// TIA Portal project "PLC2_Cell" (V19)

(* hardware
DEVICE "S7-1200 station_1"  S7-1200 Station
   slot 0: "Rack_0"  S7-1200 Rack  Rack  V1.0
   slot 1: "PLC_Machining"  CPU 1214C AC/DC/Rly  6ES7 214-1BG40-0XB0  V4.5
   slot 2: "DI 16x24VDC/DQ 16xRelay_1"  SM 1223 DI16/DQ16 x relay  6ES7 223-1PL32-0XB0  V2.0
   slot 3: "AQ 1x12BIT_1"  AQ1 signal board  6ES7 232-4HA30-0XB0  V1.0
   slot 3: "AI 4x13BIT/AQ 2x14BIT_1"  6ES7 234-4HE32-0XB0  V2.1
DEVICE "HMI_1"  KTP700 Basic PN
   slot 0: "HMI_1"  KTP700 Basic PN  6AV2 123-2GB03-0AX0  17.0.0.0
   slot 1: "HMI_RT_1"  KTP700 Basic PN  6AV2 123-2GB03-0AX0  17.0.0.0
   slot 5: "HMI_1.IE_CP_1"  PROFINET Interface  17.0.0.0
      slot 1: "PROFINET Interface_1"  PROFINET Interface
         slot 1: "Port_1"  Port
DEVICE "S7-1200 station_2"  S7-1200 Station
   slot 0: "Rack_0"  S7-1200 Rack  Rack  V1.0
   slot 1: "PLC_Pneumatic"  CPU 1214C AC/DC/Rly  6ES7 214-1BG40-0XB0  V4.5
   slot 2: "DI 16x24VDC/DQ 16xRelay_1"  SM 1223 DI16/DQ16 x relay  6ES7 223-1PL32-0XB0  V2.0
   slot 3: "AQ 1x12BIT_1"  AQ1 signal board  6ES7 232-4HA30-0XB0  V1.0
   slot 3: "AI 4x13BIT/AQ 2x14BIT_1"  6ES7 234-4HE32-0XB0  V2.1
DEVICE "HMI_2"  KTP700 Basic PN
   slot 0: "HMI_2"  KTP700 Basic PN  6AV2 123-2GB03-0AX0  17.0.0.0
   slot 1: "HMI_RT_2"  KTP700 Basic PN  6AV2 123-2GB03-0AX0  17.0.0.0
   slot 5: "HMI_2.IE_CP_1"  PROFINET Interface  17.0.0.0
      slot 1: "PROFINET Interface_1"  PROFINET Interface
         slot 1: "Port_1"  Port
*)

// ===== PLC "PLC_Machining"  CPU 1214C AC/DC/Rly =====

VAR_GLOBAL   // PLC tag table "Default tag table"
   "Pusher_latch" AT %M10.0 : Bool;
   "Conveyor2_latch" AT %M10.1 : Bool;
   "Conveyor4_latch" AT %M10.2 : Bool;
   "Conveyor3_latch" AT %M10.3 : Bool;
   "Conveyor5_latch" AT %M10.4 : Bool;
   "Conveyor6_IN_latch" AT %M10.5 : Bool;
   "Conveyor6_OUT_latch" AT %M10.6 : Bool;
   "Conveyor6_Position" AT %M10.7 : Bool;
   "lampBlinkTag" AT %M11.0 : Bool;
   "cakeFlavor" AT %MW12 : UInt;
   "drillingTime" AT %MD14 : Time;
   "mixingTime" AT %MD18 : Time;
   "System_Byte" AT %MB22 : Byte;
   "FirstScan" AT %M22.0 : Bool;
   "DiagStatusUpdate" AT %M22.1 : Bool;
   "AlwaysTRUE" AT %M22.2 : Bool;
   "AlwaysFALSE" AT %M22.3 : Bool;
   "drillActive" AT %M23.0 : Bool;
   "mixActive" AT %M23.1 : Bool;
   "CognexCode" AT %MW24 : Int;
END_VAR

VAR_GLOBAL   // PLC tag table "Cell_Tags"
   "Opto_Conveyor6B" AT %I8.0 : Bool;
   "Press_BTN_DOWN" AT %I8.2 : Bool;
   "Conveyor2" AT %Q0.0 : Bool;
   "Pusher1" AT %Q0.1 : Bool;
   "Conveyor4" AT %Q0.4 : Bool;
   "Conveyor5" AT %Q0.7 : Bool;
   "Conveyor3" AT %Q0.2 : Bool;
   "Drill" AT %Q0.3 : Bool;
   "Mix" AT %Q0.5 : Bool;
   "Pusher2" AT %Q0.6 : Bool;
   "Green_Tower" AT %Q1.0 : Bool;
   "Red_Tower" AT %Q1.1 : Bool;
   "Conveyor6_OUT" AT %Q8.3 : Bool;
   "Press_UP" AT %Q8.4 : Bool;
   "Press_DOWN" AT %Q8.5 : Bool;
   "Conveyor6_IN" AT %Q8.2 : Bool;
   "Press_BTN_UP" AT %I8.3 : Bool;
   "Opto_Conveyor2A" AT %I0.0 : Bool;
   "Opto_Conveyor2B" AT %I0.1 : Bool;
   "Green_Light" AT %Q9.5 : Bool;
   "Red_Light" AT %Q9.6 : Bool;
   "Blue_Light" AT %Q9.7 : Bool;
   "Green_BTN" AT %I9.4 : Bool;
   "Yellow_BTN" AT %I9.5 : Bool;
   "Red_BTN" AT %I9.6 : Bool;
   "Emergency_BTN" AT %I9.7 : Bool;
   "Pusher1_BTN" AT %I0.2 : Bool;
   "Opto_Drill" AT %I0.3 : Bool;
   "Opto_Mix" AT %I0.4 : Bool;
   "Opto_Conveyor5" AT %I0.6 : Bool;
   "Pusher2_BTN" AT %I0.5 : Bool;
   "Opto_Conveyor6A" AT %I8.1 : Bool;
   "Conveyor2_tactileSW" AT %I0.7 : Bool;
   "cellPotentiometer" AT %IW64 : Int;
   "AO_Channel0" AT %QW112 : Int;
   "AO_Channel1" AT %QW114 : Int;
   "AO_Cell" AT %QW80 : Int;
   "Cognex_out0" AT %I9.0 : Bool;
   "Cognex_out1" AT %I9.1 : Bool;
   "Cognex_out2" AT %I9.2 : Bool;
   "Cognex_in0" AT %Q8.7 : Bool;
END_VAR

VAR_GLOBAL   // PLC tag table "HMI_Tags"
   "HMI_BTN1" AT %M50.0 : Bool;
   "HMI_BTN_Conveyor2" AT %M50.1 : Bool;
   "HMI_BTN_Pusher1" AT %M50.2 : Bool;
   "HMI_BTN_Conveyor3" AT %M50.3 : Bool;
   "HMI_BTN_Conveyor4" AT %M50.4 : Bool;
   "HMI_BTN_Conveyor5" AT %M50.5 : Bool;
   "HMI_BTN_Drill" AT %M50.6 : Bool;
   "HMI_BTN_Mix" AT %M50.7 : Bool;
   "HMI_BTN_Pusher2" AT %M51.0 : Bool;
   "HMI_BTN10" AT %M51.1 : Bool;
   "HMI_BTN11" AT %M51.2 : Bool;
   "HMI_BTN12" AT %M51.3 : Bool;
   "HMI_BTN13" AT %M51.4 : Bool;
   "HMI_BTN14" AT %M51.5 : Bool;
   "HMI_BTN15" AT %M51.6 : Bool;
   "HMI_BTN16" AT %M51.7 : Bool;
   "HMI_BTN17" AT %M52.0 : Bool;
   "HMI_BTN18" AT %M52.1 : Bool;
   "HMI_BTN19" AT %M52.2 : Bool;
   "HMI_BTN20" AT %M52.3 : Bool;
   "HMI_BTN21" AT %M52.4 : Bool;
   "HMI_BTN22" AT %M52.5 : Bool;
   "HMI_BTN23" AT %M52.6 : Bool;
   "HMI_BTN24" AT %M52.7 : Bool;
   "ManualMode_SW" AT %M53.0 : Bool;
END_VAR

VAR_GLOBAL   // PLC tag table "Clock_Memory_Tags"
   "Clock_Byte" AT %MB0 : Byte;
   "Clock_10Hz" AT %M0.0 : Bool;
   "Clock_5Hz" AT %M0.1 : Bool;
   "Clock_2.5Hz" AT %M0.2 : Bool;
   "Clock_2Hz" AT %M0.3 : Bool;
   "Clock_1.25Hz" AT %M0.4 : Bool;
   "Clock_1Hz" AT %M0.5 : Bool;
   "Clock_0.625Hz" AT %M0.6 : Bool;
   "Clock_0.5Hz" AT %M0.7 : Bool;
END_VAR

DATA_BLOCK "potentiometerValue"   // DB14
{ S7_Optimized_Access := 'TRUE' }
VERSION : 0.1
// stored: InstanceOfName FB_AnalogInput
"FB_AnalogInput"
BEGIN
END_DATA_BLOCK

DATA_BLOCK "processTimes_DB"   // DB15
{ S7_Optimized_Access := 'TRUE' }
VERSION : 0.1
   VAR
      chocolateDrillingInput_ms : UInt := 3000;
      chocolateMixingInput_ms : UInt := 3000;
      vanillaDrillingInput_ms : UInt := 5000;
      vanillaMixingInput_ms : UInt := 5000;
      strawberryDrillingInput_ms : UInt := 7000;
      strawberryMixingInput_ms : UInt := 7000;
      chocolateDrilling_s : Time;
      chocolateMixing_s : Time;
      vanillaDrilling_s : Time;
      vanillaMixing_s : Time;
      strawberryDrilling_s : Time;
      strawberryMixing_s : Time;
   END_VAR
BEGIN
END_DATA_BLOCK

DATA_BLOCK "Machining_Communication_DB"   // DB100
{ S7_Optimized_Access := 'FALSE' }
VERSION : 0.1
   VAR
      Cognex_Code : Int;   // Machining to Pneu
      Cobot_Code : Int;   // Pneu to Machining
      Cake_ID : Int;   // Pneu to Machining
      EmergencyStop : Bool;
      Cognex_Shutter : Bool;   // Pneu to Machining
      Conveyor5_Done : Bool;   // Machining to Pneu
      Conveyor6_Done : Bool;   // Machining to Pneu
      Conveyor1_Sensor : Bool;   // Pneu to Machining
      Conveyor2_SensorA : Bool;   // Machining to Pneu
   END_VAR
BEGIN
END_DATA_BLOCK

// folder: System blocks/Program resources

DATA_BLOCK "Mix_PostTP"   // DB1
{ S7_Optimized_Access := 'TRUE' }
AUTHOR : Simatic
FAMILY : IEC
NAME : IEC_TMR
VERSION : 1.0
// stored: InstanceOfName IEC_TIMER
"IEC_TIMER"
BEGIN
END_DATA_BLOCK

DATA_BLOCK "Pusher1_Delay"   // DB2
{ S7_Optimized_Access := 'TRUE' }
AUTHOR : Simatic
FAMILY : IEC
NAME : IEC_TMR
VERSION : 1.0
// stored: InstanceOfName IEC_TIMER
"IEC_TIMER"
BEGIN
END_DATA_BLOCK

DATA_BLOCK "Drill_OperationTP"   // DB3
{ S7_Optimized_Access := 'TRUE' }
AUTHOR : Simatic
FAMILY : IEC
NAME : IEC_TMR
VERSION : 1.0
// stored: InstanceOfName IEC_TIMER
"IEC_TIMER"
BEGIN
END_DATA_BLOCK

DATA_BLOCK "Mix_OperationTP"   // DB4
{ S7_Optimized_Access := 'TRUE' }
AUTHOR : Simatic
FAMILY : IEC
NAME : IEC_TMR
VERSION : 1.0
// stored: InstanceOfName IEC_TIMER
"IEC_TIMER"
BEGIN
END_DATA_BLOCK

DATA_BLOCK "Drill_PostTP"   // DB5
{ S7_Optimized_Access := 'TRUE' }
AUTHOR : Simatic
FAMILY : IEC
NAME : IEC_TMR
VERSION : 1.0
// stored: InstanceOfName IEC_TIMER
"IEC_TIMER"
BEGIN
END_DATA_BLOCK

DATA_BLOCK "Conveyor2_TP"   // DB6
{ S7_Optimized_Access := 'TRUE' }
AUTHOR : Simatic
FAMILY : IEC
NAME : IEC_TMR
VERSION : 1.0
// stored: InstanceOfName IEC_TIMER
"IEC_TIMER"
BEGIN
END_DATA_BLOCK

DATA_BLOCK "Conveyor2_ManualDelay"   // DB7
{ S7_Optimized_Access := 'TRUE' }
AUTHOR : Simatic
FAMILY : IEC
NAME : IEC_TMR
VERSION : 1.0
// stored: InstanceOfName IEC_TIMER
"IEC_TIMER"
BEGIN
END_DATA_BLOCK

DATA_BLOCK "Pusher2_Delay"   // DB8
{ S7_Optimized_Access := 'TRUE' }
AUTHOR : Simatic
FAMILY : IEC
NAME : IEC_TMR
VERSION : 1.0
// stored: InstanceOfName IEC_TIMER
"IEC_TIMER"
BEGIN
END_DATA_BLOCK

DATA_BLOCK "Press_Delay"   // DB9
{ S7_Optimized_Access := 'TRUE' }
AUTHOR : Simatic
FAMILY : IEC
NAME : IEC_TMR
VERSION : 1.0
// stored: InstanceOfName IEC_TIMER
"IEC_TIMER"
BEGIN
END_DATA_BLOCK

DATA_BLOCK "IEC_Timer_0_DB"   // DB10
{ S7_Optimized_Access := 'TRUE' }
AUTHOR : Simatic
FAMILY : IEC
NAME : IEC_TMR
VERSION : 1.0
// stored: InstanceOfName IEC_TIMER
"IEC_TIMER"
BEGIN
END_DATA_BLOCK

DATA_BLOCK "Press_DOWN_Timer"   // DB11
{ S7_Optimized_Access := 'TRUE' }
AUTHOR : Simatic
FAMILY : IEC
NAME : IEC_TMR
VERSION : 1.0
// stored: InstanceOfName IEC_TIMER
"IEC_TIMER"
BEGIN
END_DATA_BLOCK

DATA_BLOCK "Emergency_Blink_TP"   // DB12
{ S7_Optimized_Access := 'TRUE' }
AUTHOR : Simatic
FAMILY : IEC
NAME : IEC_TMR
VERSION : 1.0
// stored: InstanceOfName IEC_TIMER
"IEC_TIMER"
BEGIN
END_DATA_BLOCK

DATA_BLOCK "Emergency_Blink_TON"   // DB13
{ S7_Optimized_Access := 'TRUE' }
AUTHOR : Simatic
FAMILY : IEC
NAME : IEC_TMR
VERSION : 1.0
// stored: InstanceOfName IEC_TIMER
"IEC_TIMER"
BEGIN
END_DATA_BLOCK

// folder: (top level)

FUNCTION_BLOCK "FB_AnalogInput"   // FB1, LAD
{ S7_Optimized_Access := 'TRUE' }
VERSION : 0.1
   VAR_INPUT
      minRaw : Int;
      maxRaw : Int := 27648;
      rawValue : Int;
      minScale : Real;
      maxScale : Real := 1.0;
   END_VAR
   VAR_OUTPUT
      outputValue : Real;
   END_VAR
   VAR_TEMP
      normValue : Real;
   END_VAR
BEGIN

REGION Network 1
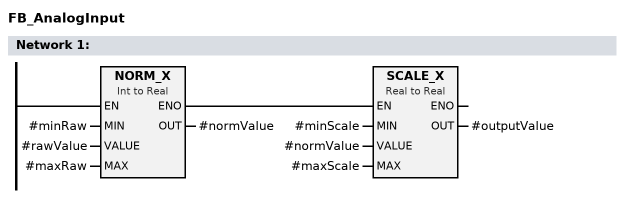
   RUNG wire#powerrail
      { S7_Templates := "[SrcType := Int, DestType := Real]" } Normalize(min := #minRaw, value := #rawValue, max := #maxRaw, out => #normValue)
      { S7_Templates := "[SrcType := Real, DestType := Real]" } Scale(min := #minScale, value := #normValue, max := #maxScale, out => #outputValue)
   END_RUNG
   // the same network as SCL:
   #normValue := NORM_X(MIN := #minRaw, VALUE := #rawValue, MAX := #maxRaw);
   #outputValue := SCALE_X(MIN := #minScale, VALUE := #normValue, MAX := #maxScale);
END_REGION
END_FUNCTION_BLOCK

ORGANIZATION_BLOCK "Main"   // OB1, LAD, ProgramCycle
TITLE = "Main Program Sweep (Cycle)"
{ S7_Optimized_Access := 'TRUE' }
VERSION : 0.1
   VAR_INPUT
      Initial_Call : Bool;   // Initial call of this OB
      Remanence : Bool;   // =True, if remanent data are available
   END_VAR
   VAR_TEMP   // added for the SCL form of the ladder/FBD networks
      _w1 : Bool;
   END_VAR
BEGIN

REGION Network 1: Conveyor #2
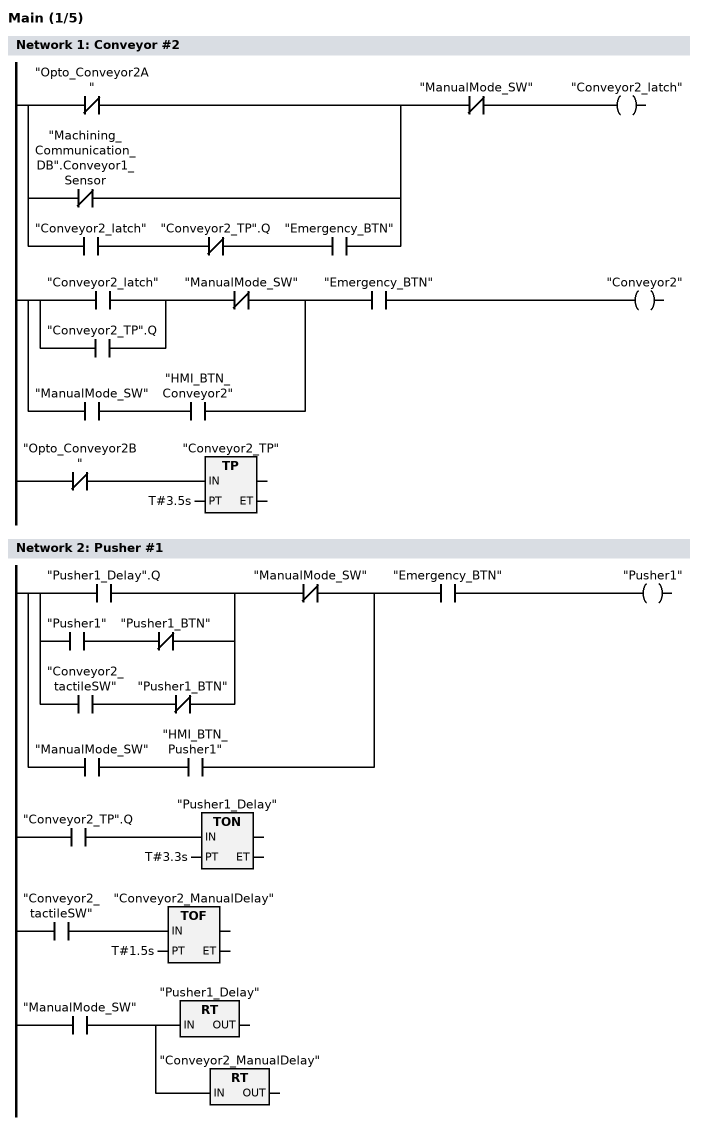
   "Conveyor2_latch" := (NOT "Opto_Conveyor2A" OR NOT "Machining_Communication_DB".Conveyor1_Sensor OR ("Conveyor2_latch" AND NOT "Conveyor2_TP".Q AND "Emergency_BTN")) AND NOT "ManualMode_SW";
   "Conveyor2" := ((("Conveyor2_latch" OR "Conveyor2_TP".Q) AND NOT "ManualMode_SW") OR ("ManualMode_SW" AND "HMI_BTN_Conveyor2")) AND "Emergency_BTN";
   "Conveyor2_TP".TP(IN := NOT "Opto_Conveyor2B", PT := T#3.5s);
END_REGION

REGION Network 2: Pusher #1
   "Pusher1" := ((("Pusher1_Delay".Q OR ("Pusher1" AND NOT "Pusher1_BTN") OR ("Conveyor2_tactileSW" AND NOT "Pusher1_BTN")) AND NOT "ManualMode_SW") OR ("ManualMode_SW" AND "HMI_BTN_Pusher1")) AND "Emergency_BTN";
   "Pusher1_Delay".TON(IN := "Conveyor2_TP".Q, PT := T#3.3s);
   "Conveyor2_ManualDelay".TOF(IN := "Conveyor2_tactileSW", PT := T#1.5s);
   IF "ManualMode_SW" THEN
       RESET_TIMER("Pusher1_Delay");
       RESET_TIMER("Conveyor2_ManualDelay");
   END_IF;
END_REGION

REGION Network 3: Conveyor 3: Drill
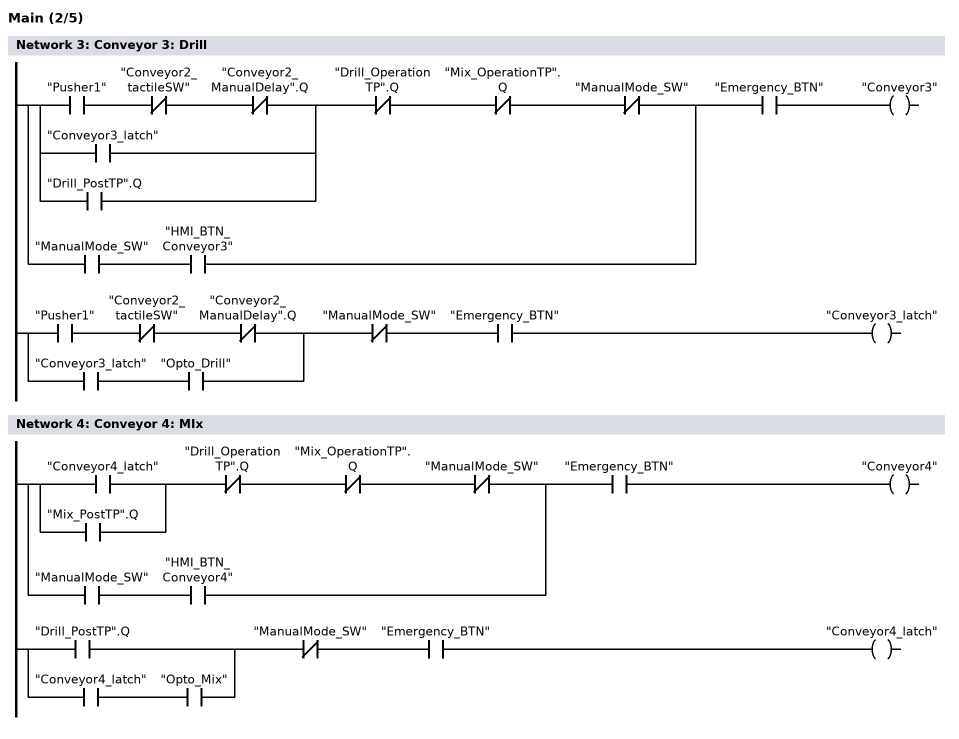
   RUNG wire#powerrail
      Contact( "Pusher1" )
      I_Contact( "Conveyor2_tactileSW" )
      I_Contact( "Conveyor2_ManualDelay".Q )
      wire#w1
      I_Contact( "Drill_OperationTP".Q )
      I_Contact( "Mix_OperationTP".Q )
      I_Contact( "ManualMode_SW" )
      wire#w2
      Contact( "Emergency_BTN" )
      Coil( "Conveyor3" )
   END_RUNG
   RUNG wire#powerrail
      Contact( "Conveyor3_latch" )
   END_RUNG wire#w1
   RUNG wire#powerrail
      Contact( "Drill_PostTP".Q )
   END_RUNG wire#w1
   RUNG wire#powerrail
      Contact( "ManualMode_SW" )
      Contact( "HMI_BTN_Conveyor3" )
   END_RUNG wire#w2
   RUNG wire#powerrail
      Contact( "Pusher1" )
      I_Contact( "Conveyor2_tactileSW" )
      I_Contact( "Conveyor2_ManualDelay".Q )
      wire#w3
      I_Contact( "ManualMode_SW" )
      Contact( "Emergency_BTN" )
      Coil( "Conveyor3_latch" )
   END_RUNG
   RUNG wire#powerrail
      Contact( "Conveyor3_latch" )
      Contact( "Opto_Drill" )
   END_RUNG wire#w3
   // the same network as SCL:
   "Conveyor3" := (((("Pusher1" AND NOT "Conveyor2_tactileSW" AND NOT "Conveyor2_ManualDelay".Q) OR "Conveyor3_latch" OR "Drill_PostTP".Q) AND NOT "Drill_OperationTP".Q AND NOT "Mix_OperationTP".Q AND NOT "ManualMode_SW") OR ("ManualMode_SW" AND "HMI_BTN_Conveyor3")) AND "Emergency_BTN";
   "Conveyor3_latch" := (("Pusher1" AND NOT "Conveyor2_tactileSW" AND NOT "Conveyor2_ManualDelay".Q) OR ("Conveyor3_latch" AND "Opto_Drill")) AND NOT "ManualMode_SW" AND "Emergency_BTN";
END_REGION

REGION Network 4: Conveyor 4: MIx
   RUNG wire#powerrail
      Contact( "Conveyor4_latch" )
      wire#w1
      I_Contact( "Drill_OperationTP".Q )
      I_Contact( "Mix_OperationTP".Q )
      I_Contact( "ManualMode_SW" )
      wire#w2
      Contact( "Emergency_BTN" )
      Coil( "Conveyor4" )
   END_RUNG
   RUNG wire#powerrail
      Contact( "Mix_PostTP".Q )
   END_RUNG wire#w1
   RUNG wire#powerrail
      Contact( "ManualMode_SW" )
      Contact( "HMI_BTN_Conveyor4" )
   END_RUNG wire#w2
   RUNG wire#powerrail
      Contact( "Drill_PostTP".Q )
      wire#w3
      I_Contact( "ManualMode_SW" )
      Contact( "Emergency_BTN" )
      Coil( "Conveyor4_latch" )
   END_RUNG
   RUNG wire#powerrail
      Contact( "Conveyor4_latch" )
      Contact( "Opto_Mix" )
   END_RUNG wire#w3
   // the same network as SCL:
   "Conveyor4" := ((("Conveyor4_latch" OR "Mix_PostTP".Q) AND NOT "Drill_OperationTP".Q AND NOT "Mix_OperationTP".Q AND NOT "ManualMode_SW") OR ("ManualMode_SW" AND "HMI_BTN_Conveyor4")) AND "Emergency_BTN";
   "Conveyor4_latch" := ("Drill_PostTP".Q OR ("Conveyor4_latch" AND "Opto_Mix")) AND NOT "ManualMode_SW" AND "Emergency_BTN";
END_REGION

REGION Network 5: Drill and Mix
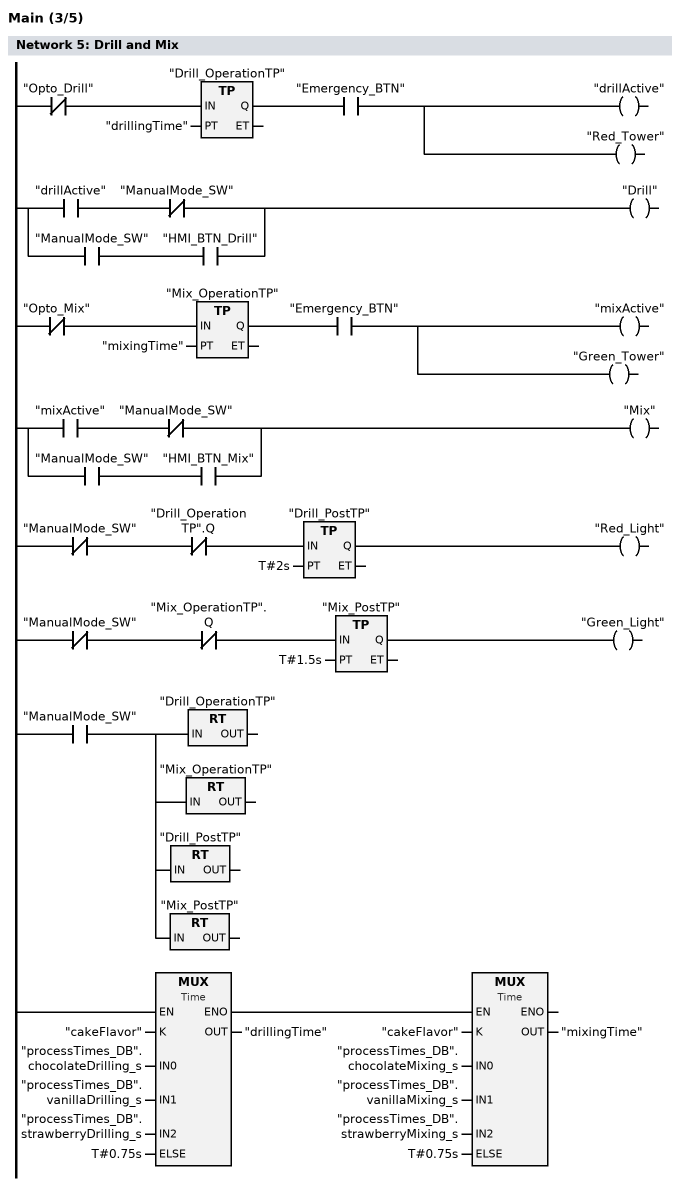
   // no SCL statement known for Mux: written as a call
   // ENO of a box is taken as its EN; it also drops when the box reports an error
   "Drill_OperationTP".TP(IN := NOT "Opto_Drill", PT := "drillingTime");
   "drillActive" := "Drill_OperationTP".Q AND "Emergency_BTN";
   "Red_Tower" := "drillActive";
   "Drill" := ("drillActive" AND NOT "ManualMode_SW") OR ("ManualMode_SW" AND "HMI_BTN_Drill");
   "Mix_OperationTP".TP(IN := NOT "Opto_Mix", PT := "mixingTime");
   "mixActive" := "Mix_OperationTP".Q AND "Emergency_BTN";
   "Green_Tower" := "mixActive";
   "Mix" := ("mixActive" AND NOT "ManualMode_SW") OR ("ManualMode_SW" AND "HMI_BTN_Mix");
   "Drill_PostTP".TP(IN := NOT "ManualMode_SW" AND NOT "Drill_OperationTP".Q, PT := T#2s);
   "Red_Light" := "Drill_PostTP".Q;
   "Mix_PostTP".TP(IN := NOT "ManualMode_SW" AND NOT "Mix_OperationTP".Q, PT := T#1.5s);
   "Green_Light" := "Mix_PostTP".Q;
   IF "ManualMode_SW" THEN
       RESET_TIMER("Drill_OperationTP");
       RESET_TIMER("Mix_OperationTP");
       RESET_TIMER("Drill_PostTP");
       RESET_TIMER("Mix_PostTP");
   END_IF;
   Mux(k := "cakeFlavor",
       in0 := "processTimes_DB".chocolateDrilling_s,
       in1 := "processTimes_DB".vanillaDrilling_s,
       in2 := "processTimes_DB".strawberryDrilling_s,
       "else" := T#0.75s,
       out => "drillingTime");
   Mux(k := "cakeFlavor",
       in0 := "processTimes_DB".chocolateMixing_s,
       in1 := "processTimes_DB".vanillaMixing_s,
       in2 := "processTimes_DB".strawberryMixing_s,
       "else" := T#0.75s,
       out => "mixingTime");
END_REGION

REGION Network 6: Pusher #2
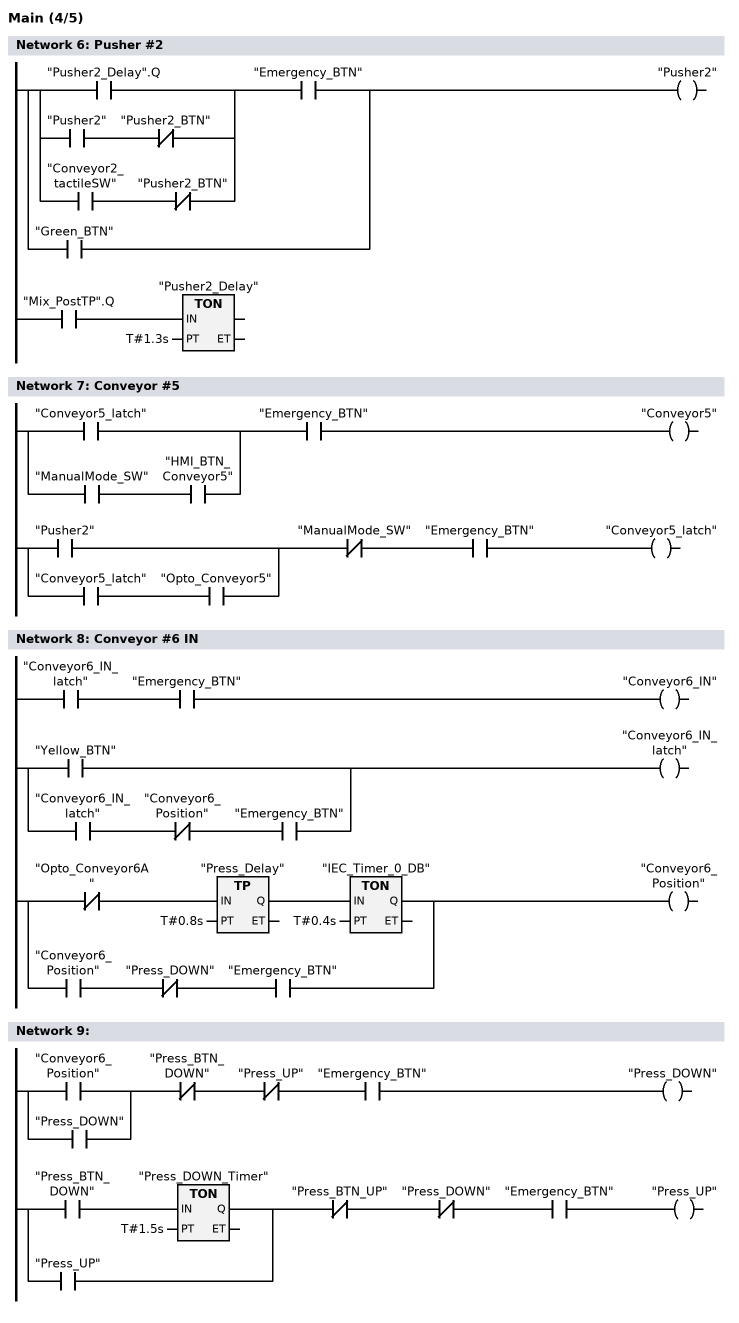
   "Pusher2" := (("Pusher2_Delay".Q OR ("Pusher2" AND NOT "Pusher2_BTN") OR ("Conveyor2_tactileSW" AND NOT "Pusher2_BTN")) AND "Emergency_BTN") OR "Green_BTN";
   "Pusher2_Delay".TON(IN := "Mix_PostTP".Q, PT := T#1.3s);
END_REGION

REGION Network 7: Conveyor #5
   RUNG wire#powerrail
      Contact( "Conveyor5_latch" )
      wire#w1
      Contact( "Emergency_BTN" )
      Coil( "Conveyor5" )
   END_RUNG
   RUNG wire#powerrail
      Contact( "ManualMode_SW" )
      Contact( "HMI_BTN_Conveyor5" )
   END_RUNG wire#w1
   RUNG wire#powerrail
      Contact( "Pusher2" )
      wire#w2
      I_Contact( "ManualMode_SW" )
      Contact( "Emergency_BTN" )
      Coil( "Conveyor5_latch" )
   END_RUNG
   RUNG wire#powerrail
      Contact( "Conveyor5_latch" )
      Contact( "Opto_Conveyor5" )
   END_RUNG wire#w2
   // the same network as SCL:
   "Conveyor5" := ("Conveyor5_latch" OR ("ManualMode_SW" AND "HMI_BTN_Conveyor5")) AND "Emergency_BTN";
   "Conveyor5_latch" := ("Pusher2" OR ("Conveyor5_latch" AND "Opto_Conveyor5")) AND NOT "ManualMode_SW" AND "Emergency_BTN";
END_REGION

REGION Network 8: Conveyor #6 IN
   "Conveyor6_IN" := "Conveyor6_IN_latch" AND "Emergency_BTN";
   "Conveyor6_IN_latch" := "Yellow_BTN" OR ("Conveyor6_IN_latch" AND NOT "Conveyor6_Position" AND "Emergency_BTN");
   "Press_Delay".TP(IN := NOT "Opto_Conveyor6A", PT := T#0.8s);
   "IEC_Timer_0_DB".TON(IN := "Press_Delay".Q, PT := T#0.4s);
   "Conveyor6_Position" := "IEC_Timer_0_DB".Q OR ("Conveyor6_Position" AND NOT "Press_DOWN" AND "Emergency_BTN");
END_REGION

REGION Network 9
   "Press_DOWN" := ("Conveyor6_Position" OR "Press_DOWN") AND NOT "Press_BTN_DOWN" AND NOT "Press_UP" AND "Emergency_BTN";
   "Press_DOWN_Timer".TON(IN := "Press_BTN_DOWN", PT := T#1.5s);
   "Press_UP" := ("Press_DOWN_Timer".Q OR "Press_UP") AND NOT "Press_BTN_UP" AND NOT "Press_DOWN" AND "Emergency_BTN";
END_REGION

REGION Network 10: Conveyor #6 OUT
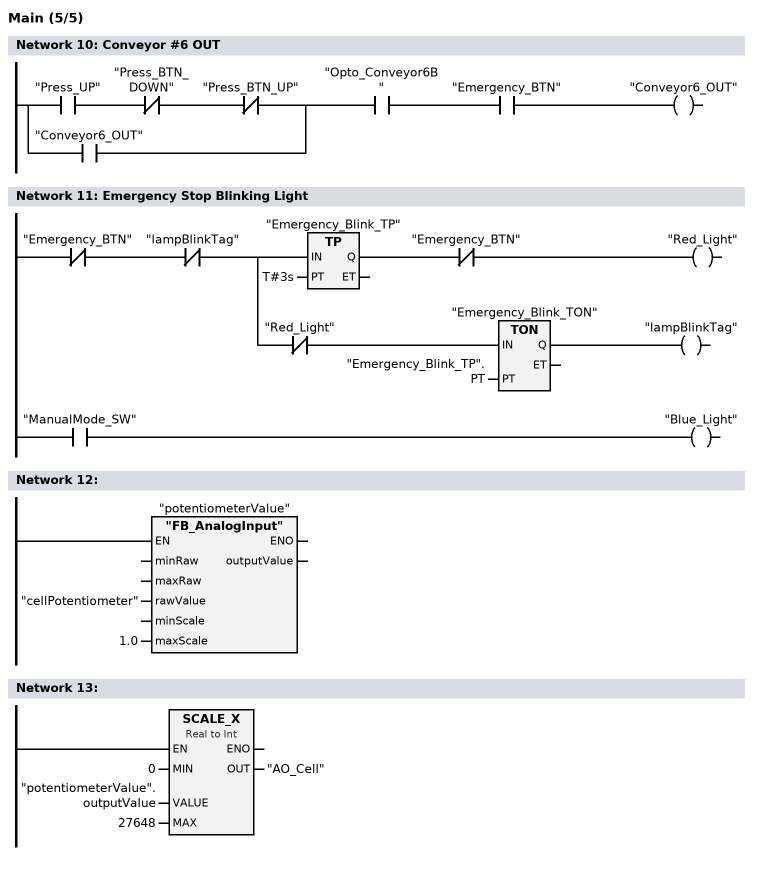
   RUNG wire#powerrail
      Contact( "Press_UP" )
      I_Contact( "Press_BTN_DOWN" )
      I_Contact( "Press_BTN_UP" )
      wire#w1
      Contact( "Opto_Conveyor6B" )
      Contact( "Emergency_BTN" )
      Coil( "Conveyor6_OUT" )
   END_RUNG
   RUNG wire#powerrail
      Contact( "Conveyor6_OUT" )
   END_RUNG wire#w1
   // the same network as SCL:
   "Conveyor6_OUT" := (("Press_UP" AND NOT "Press_BTN_DOWN" AND NOT "Press_BTN_UP") OR "Conveyor6_OUT") AND "Opto_Conveyor6B" AND "Emergency_BTN";
END_REGION

REGION Network 11: Emergency Stop Blinking Light
   #_w1 := NOT "Emergency_BTN" AND NOT "lampBlinkTag";
   "Emergency_Blink_TP".TP(IN := #_w1, PT := T#3s);
   "Red_Light" := "Emergency_Blink_TP".Q AND NOT "Emergency_BTN";
   "Emergency_Blink_TON".TON(IN := #_w1 AND NOT "Red_Light", PT := "Emergency_Blink_TP".PT);
   "lampBlinkTag" := "Emergency_Blink_TON".Q;
   "Blue_Light" := "ManualMode_SW";
END_REGION

REGION Network 12
   RUNG wire#powerrail
      "potentiometerValue"(minRaw :=, maxRaw :=, rawValue := "cellPotentiometer", minScale :=, maxScale := 1.0, outputValue =>)
   END_RUNG
   // the same network as SCL:
   "potentiometerValue"(rawValue := "cellPotentiometer", maxScale := 1.0);   // "FB_AnalogInput"
END_REGION

REGION Network 13
   RUNG wire#powerrail
      { S7_Templates := "[SrcType := Real, DestType := Int]" } Scale(min := 0, value := "potentiometerValue".outputValue, max := 27648, out => "AO_Cell")
   END_RUNG
   // the same network as SCL:
   "AO_Cell" := SCALE_X(MIN := 0, VALUE := "potentiometerValue".outputValue, MAX := 27648);
END_REGION
END_ORGANIZATION_BLOCK

ORGANIZATION_BLOCK "HMI_OB"   // OB123, LAD, ProgramCycle
TITLE = "Main Program Sweep (Cycle)"
{ S7_Optimized_Access := 'TRUE' }
VERSION : 0.1
   VAR_INPUT
      Initial_Call : Bool;   // Initial call of this OB
      Remanence : Bool;   // =True, if remanent data are available
   END_VAR
BEGIN

REGION Network 1
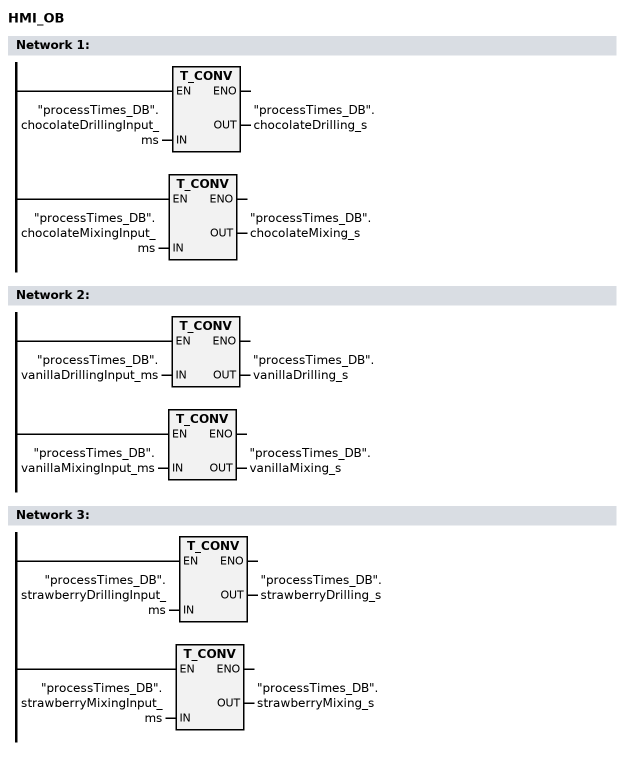
   "processTimes_DB".chocolateDrilling_s := T_CONV(IN := "processTimes_DB".chocolateDrillingInput_ms);
   "processTimes_DB".chocolateMixing_s := T_CONV(IN := "processTimes_DB".chocolateMixingInput_ms);
END_REGION

REGION Network 2
   "processTimes_DB".vanillaDrilling_s := T_CONV(IN := "processTimes_DB".vanillaDrillingInput_ms);
   "processTimes_DB".vanillaMixing_s := T_CONV(IN := "processTimes_DB".vanillaMixingInput_ms);
END_REGION

REGION Network 3
   "processTimes_DB".strawberryDrilling_s := T_CONV(IN := "processTimes_DB".strawberryDrillingInput_ms);
   "processTimes_DB".strawberryMixing_s := T_CONV(IN := "processTimes_DB".strawberryMixingInput_ms);
END_REGION
END_ORGANIZATION_BLOCK

ORGANIZATION_BLOCK "Cognex_OB"   // OB124, LAD, ProgramCycle
TITLE = "Main Program Sweep (Cycle)"
{ S7_Optimized_Access := 'TRUE' }
VERSION : 0.1
   VAR_INPUT
      Initial_Call : Bool;   // Initial call of this OB
      Remanence : Bool;   // =True, if remanent data are available
   END_VAR
BEGIN

REGION Network 1
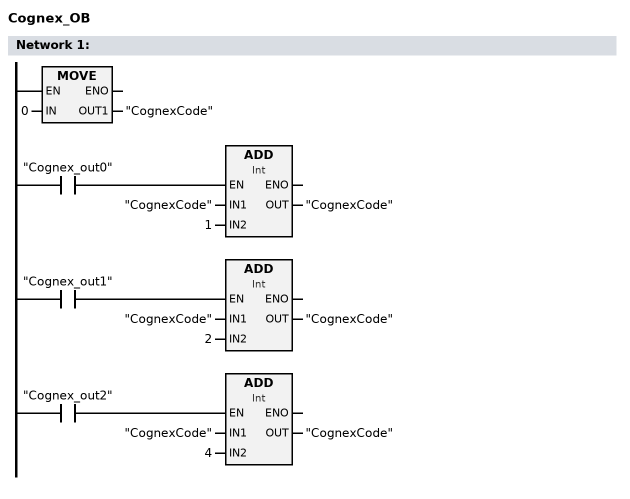
   RUNG wire#powerrail
      Move(in := 0, out1 => "CognexCode")
   END_RUNG
   RUNG wire#powerrail
      Contact( "Cognex_out0" )
      { S7_Templates := "SrcType := Int" } Add(in1 := "CognexCode", in2 := 1, out => "CognexCode")
   END_RUNG
   RUNG wire#powerrail
      Contact( "Cognex_out1" )
      { S7_Templates := "SrcType := Int" } Add(in1 := "CognexCode", in2 := 2, out => "CognexCode")
   END_RUNG
   RUNG wire#powerrail
      Contact( "Cognex_out2" )
      { S7_Templates := "SrcType := Int" } Add(in1 := "CognexCode", in2 := 4, out => "CognexCode")
   END_RUNG
   // the same network as SCL:
   "CognexCode" := 0;
   IF "Cognex_out0" THEN "CognexCode" := "CognexCode" + 1; END_IF;
   IF "Cognex_out1" THEN "CognexCode" := "CognexCode" + 2; END_IF;
   IF "Cognex_out2" THEN "CognexCode" := "CognexCode" + 4; END_IF;
END_REGION
END_ORGANIZATION_BLOCK

// ===== PLC "PLC_Pneumatic"  CPU 1214C AC/DC/Rly =====

VAR_GLOBAL   // PLC tag table "Default tag table"
   "normPressure" AT %MD30 : Real;
   "pressureValue" AT %MD34 : Real;
   "cakeFlavor" AT %MW38 : UInt;
   "PunchingTime" AT %MD40 : Time;
END_VAR

VAR_GLOBAL   // PLC tag table "Cell_Tags"
   "Red_BTN" AT %I9.6 : Bool;
   "Green_BTN" AT %I9.4 : Bool;
   "Yellow_BTN" AT %I9.5 : Bool;
   "Emergency_BTN" AT %I9.7 : Bool;
   "Opto_Start" AT %I8.0 : Bool;
   "Vertical_Punch_BTN" AT %I8.1 : Bool;
   "Turntable_BTN" AT %I8.3 : Bool;
   "In_Conveyor_BTN" AT %I8.4 : Bool;
   "Red_Light" AT %Q9.6 : Bool;
   "Green_Light" AT %Q9.5 : Bool;
   "Blue_Light" AT %Q9.7 : Bool;
   "Turntable" AT %Q9.0 : Bool;
   "Conveyor1" AT %Q9.1 : Bool;
   "Ext_Piston_Start" AT %Q8.4 : Bool;
   "Cntrcn_Piston_Start" AT %Q8.3 : Bool;
   "Vertical_Piston" AT %Q8.5 : Bool;
   "Ext_Piston_Conveyor" AT %Q8.7 : Bool;
   "Cntrcn_Piston_Conveyor" AT %Q8.6 : Bool;
   "Opto_Conveyor_Exit1" AT %I8.5 : Bool;
   "pressureSensor" AT %IW118 : Int;
END_VAR

VAR_GLOBAL   // PLC tag table "Cobot_Tags"
   "Stop_Moving_Cobot" AT %Q8.0 : Bool;
   "Cobot_Moving" AT %I0.0 : Bool;
   "Cobot_DI_1" AT %Q8.1 : Bool;
   "Cobot_DI_2" AT %Q8.2 : Bool;
   "Cobot_DI_3" AT %Q9.4 : Bool;
   "Cobot_DO_1" AT %I0.1 : Bool;
   "Cobot_DO_2" AT %I0.2 : Bool;
   "Cobot_DO_3" AT %I0.3 : Bool;
END_VAR

VAR_GLOBAL   // PLC tag table "HMI_Tags"
   "Green_BTN_HMI" AT %M20.0 : Bool;
   "Yellow_BTN_HMI" AT %M20.1 : Bool;
   "Red_BTN_HMI" AT %M20.2 : Bool;
   "Cntrcn_Piston_Conveyor_HMI" AT %M20.3 : Bool;
   "Vertical_Piston_HMI" AT %M20.4 : Bool;
   "Cntrcn_Piston_Start_HMI" AT %M20.5 : Bool;
   "Ext_Piston_Start_HMI" AT %M20.6 : Bool;
   "Ext_Piston_Conveyor_HMI" AT %M20.7 : Bool;
   "Conveyor1_HMI" AT %M21.0 : Bool;
   "Turntable_HMI" AT %M21.1 : Bool;
END_VAR

VAR_GLOBAL   // PLC tag table "Clock_Memory_Tags"
   "Clock_Byte" AT %MB0 : Byte;
   "Clock_10Hz" AT %M0.0 : Bool;
   "Clock_5Hz" AT %M0.1 : Bool;
   "Clock_2.5Hz" AT %M0.2 : Bool;
   "Clock_2Hz" AT %M0.3 : Bool;
   "Clock_1.25Hz" AT %M0.4 : Bool;
   "Clock_1Hz" AT %M0.5 : Bool;
   "Clock_0.625Hz" AT %M0.6 : Bool;
   "Clock_0.5Hz" AT %M0.7 : Bool;
END_VAR

DATA_BLOCK "Pneumatic_Times_DB"   // DB20
{ S7_Optimized_Access := 'TRUE' }
VERSION : 0.1
   VAR
      chocolatePunchingInput_ms : UInt := 2000;
      vanillaPunchingInput_ms : UInt := 4000;
      strawberryPunchingInput_ms : UInt := 6000;
      chocolatePunching_s : Time;
      vanillaPunching_s : Time;
      strawberryPunching_s : Time;
   END_VAR
BEGIN
END_DATA_BLOCK

DATA_BLOCK "Pneumatic_Communication_DB"   // DB100
{ S7_Optimized_Access := 'FALSE' }
VERSION : 0.1
   VAR
      Cognex_Code : Int;
      Cobot_Code : Int;
      Cake_ID : Int;
      EmergencyStop : Bool;
      Cognex_Shutter : Bool;
      Conveyor5_Done : Bool;
      Conveyor6_Done : Bool;
      Conveyor1_Sensor : Bool;
      Conveyor2_SensorA : Bool;
   END_VAR
BEGIN
END_DATA_BLOCK

// folder: System blocks/Program resources

DATA_BLOCK "TON_Start"   // DB1
{ S7_Optimized_Access := 'TRUE' }
AUTHOR : Simatic
FAMILY : IEC
NAME : IEC_TMR
VERSION : 1.0
// stored: InstanceOfName IEC_TIMER
"IEC_TIMER"
BEGIN
END_DATA_BLOCK

DATA_BLOCK "TOF_Start"   // DB2
{ S7_Optimized_Access := 'TRUE' }
AUTHOR : Simatic
FAMILY : IEC
NAME : IEC_TMR
VERSION : 1.0
// stored: InstanceOfName IEC_TIMER
"IEC_TIMER"
BEGIN
END_DATA_BLOCK

DATA_BLOCK "TON_vertical_piston"   // DB4
{ S7_Optimized_Access := 'TRUE' }
AUTHOR : Simatic
FAMILY : IEC
NAME : IEC_TMR
VERSION : 1.0
// stored: InstanceOfName IEC_TIMER
"IEC_TIMER"
BEGIN
END_DATA_BLOCK

DATA_BLOCK "TON_Turntable"   // DB5
{ S7_Optimized_Access := 'TRUE' }
AUTHOR : Simatic
FAMILY : IEC
NAME : IEC_TMR
VERSION : 1.0
// stored: InstanceOfName IEC_TIMER
"IEC_TIMER"
BEGIN
END_DATA_BLOCK

DATA_BLOCK "TP_piston_in_conveyor"   // DB6
{ S7_Optimized_Access := 'TRUE' }
AUTHOR : Simatic
FAMILY : IEC
NAME : IEC_TMR
VERSION : 1.0
// stored: InstanceOfName IEC_TIMER
"IEC_TIMER"
BEGIN
END_DATA_BLOCK

// folder: (top level)

ORGANIZATION_BLOCK "Main"   // OB1, LAD, ProgramCycle
TITLE = "Main Program Sweep (Cycle)"
{ S7_Optimized_Access := 'TRUE' }
VERSION : 0.1
   VAR_INPUT
      Initial_Call : Bool;   // Initial call of this OB
      Remanence : Bool;   // =True, if remanent data are available
   END_VAR
BEGIN

REGION Network 1: Punching time multiplexer
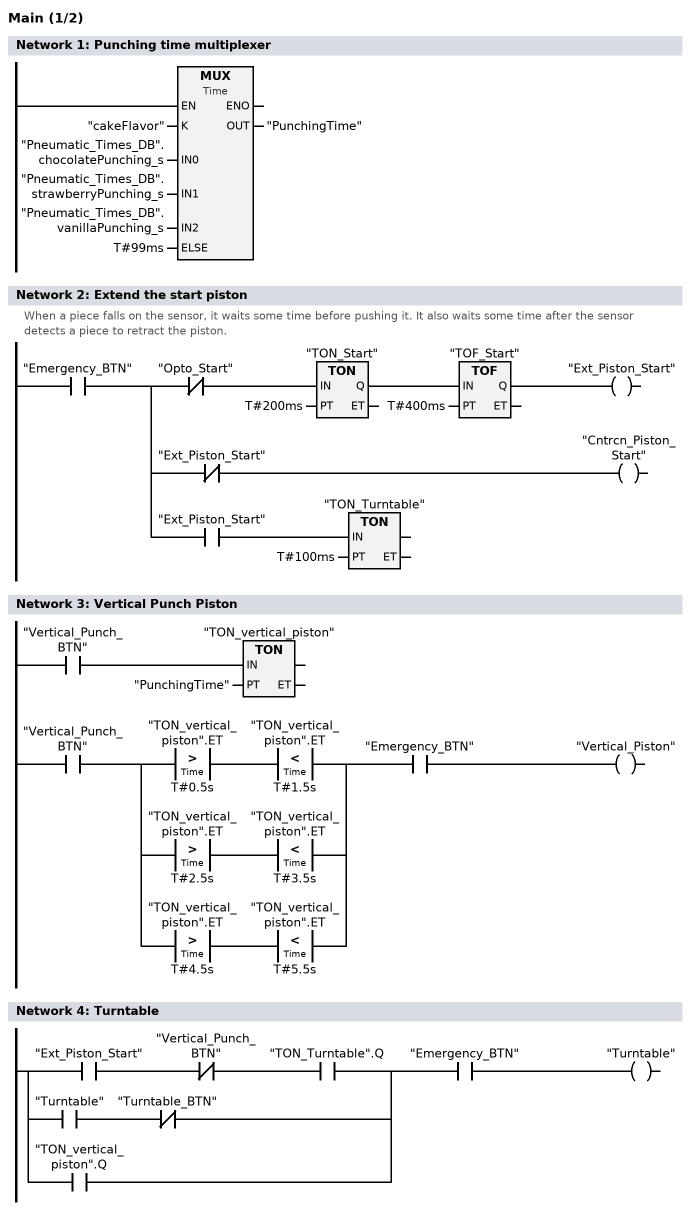
   RUNG wire#powerrail
      { S7_Templates := "SrcType := Time"; S7_GenerateENO := "TRUE" } Mux(k := "cakeFlavor", in0 := "Pneumatic_Times_DB".chocolatePunching_s, in1 := "Pneumatic_Times_DB".strawberryPunching_s, in2 := "Pneumatic_Times_DB".vanillaPunching_s, "else" := T#99ms, out => "PunchingTime")
   END_RUNG
   // the same network as SCL:
   // no SCL statement known for Mux: written as a call
   Mux(k := "cakeFlavor",
       in0 := "Pneumatic_Times_DB".chocolatePunching_s,
       in1 := "Pneumatic_Times_DB".strawberryPunching_s,
       in2 := "Pneumatic_Times_DB".vanillaPunching_s,
       "else" := T#99ms,
       out => "PunchingTime");
END_REGION

REGION Network 2: Extend the start piston
   // When a piece falls on the sensor, it waits some time before pushing it. It also waits some time after the sensor detects a piece to retract the piston.
   "TON_Start".TON(IN := "Emergency_BTN" AND NOT "Opto_Start", PT := T#200ms);
   "TOF_Start".TOF(IN := "TON_Start".Q, PT := T#400ms);
   "Ext_Piston_Start" := "TOF_Start".Q;
   "Cntrcn_Piston_Start" := "Emergency_BTN" AND NOT "Ext_Piston_Start";
   "TON_Turntable".TON(IN := "Emergency_BTN" AND "Ext_Piston_Start", PT := T#100ms);
END_REGION

REGION Network 3: Vertical Punch Piston
   "TON_vertical_piston".TON(IN := "Vertical_Punch_BTN", PT := "PunchingTime");
   "Vertical_Piston" := "Vertical_Punch_BTN" AND ((("TON_vertical_piston".ET > T#0.5s) AND ("TON_vertical_piston".ET < T#1.5s)) OR (("TON_vertical_piston".ET > T#2.5s) AND ("TON_vertical_piston".ET < T#3.5s)) OR (("TON_vertical_piston".ET > T#4.5s) AND ("TON_vertical_piston".ET < T#5.5s))) AND "Emergency_BTN";
END_REGION

REGION Network 4: Turntable
   RUNG wire#powerrail
      Contact( "Ext_Piston_Start" )
      I_Contact( "Vertical_Punch_BTN" )
      Contact( "TON_Turntable".Q )
      wire#w1
      Contact( "Emergency_BTN" )
      Coil( "Turntable" )
   END_RUNG
   RUNG wire#powerrail
      Contact( "Turntable" )
      I_Contact( "Turntable_BTN" )
   END_RUNG wire#w1
   RUNG wire#powerrail
      Contact( "TON_vertical_piston".Q )
   END_RUNG wire#w1
   // the same network as SCL:
   "Turntable" := (("Ext_Piston_Start" AND NOT "Vertical_Punch_BTN" AND "TON_Turntable".Q) OR ("Turntable" AND NOT "Turntable_BTN") OR "TON_vertical_piston".Q) AND "Emergency_BTN";
END_REGION

REGION Network 5: Piston Conveyor
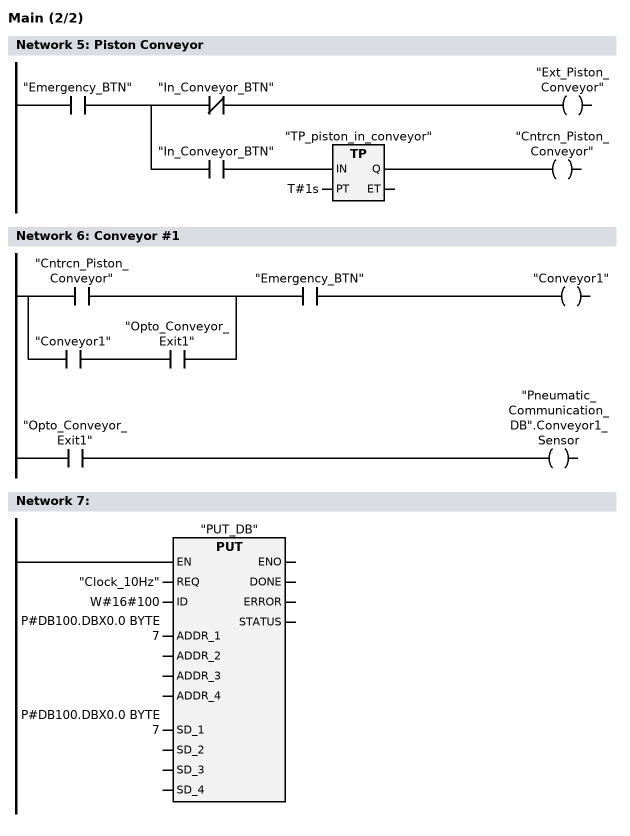
   "Ext_Piston_Conveyor" := "Emergency_BTN" AND NOT "In_Conveyor_BTN";
   "TP_piston_in_conveyor".TP(IN := "Emergency_BTN" AND "In_Conveyor_BTN", PT := T#1s);
   "Cntrcn_Piston_Conveyor" := "TP_piston_in_conveyor".Q;
END_REGION

REGION Network 6: Conveyor #1
   RUNG wire#powerrail
      Contact( "Cntrcn_Piston_Conveyor" )
      wire#w1
      Contact( "Emergency_BTN" )
      Coil( "Conveyor1" )
   END_RUNG
   RUNG wire#powerrail
      Contact( "Conveyor1" )
      Contact( "Opto_Conveyor_Exit1" )
   END_RUNG wire#w1
   RUNG wire#powerrail
      Contact( "Opto_Conveyor_Exit1" )
      Coil( "Pneumatic_Communication_DB".Conveyor1_Sensor )
   END_RUNG
   // the same network as SCL:
   "Conveyor1" := ("Cntrcn_Piston_Conveyor" OR ("Conveyor1" AND "Opto_Conveyor_Exit1")) AND "Emergency_BTN";
   "Pneumatic_Communication_DB".Conveyor1_Sensor := "Opto_Conveyor_Exit1";
END_REGION

REGION Network 7
   "PUT_DB"(REQ := "Clock_10Hz", ID := W#16#100, ADDR_1 := P#DB100.DBX0.0 BYTE 7, SD_1 := P#DB100.DBX0.0 BYTE 7);   // PUT
END_REGION
END_ORGANIZATION_BLOCK

ORGANIZATION_BLOCK "HMI_OB"   // OB123, LAD, ProgramCycle
TITLE = "Main Program Sweep (Cycle)"
{ S7_Optimized_Access := 'TRUE' }
VERSION : 0.1
   VAR_INPUT
      Initial_Call : Bool;   // Initial call of this OB
      Remanence : Bool;   // =True, if remanent data are available
   END_VAR
BEGIN

REGION Network 1
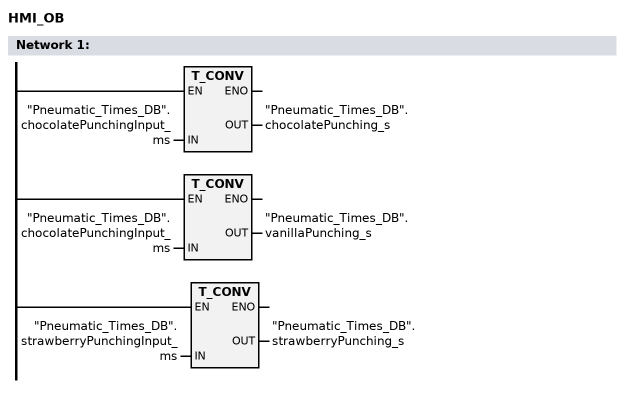
   "Pneumatic_Times_DB".chocolatePunching_s := T_CONV(IN := "Pneumatic_Times_DB".chocolatePunchingInput_ms);
   "Pneumatic_Times_DB".vanillaPunching_s := T_CONV(IN := "Pneumatic_Times_DB".chocolatePunchingInput_ms);
   "Pneumatic_Times_DB".strawberryPunching_s := T_CONV(IN := "Pneumatic_Times_DB".strawberryPunchingInput_ms);
END_REGION
END_ORGANIZATION_BLOCK

ORGANIZATION_BLOCK "Cobot_OB"   // OB124, LAD, ProgramCycle
TITLE = "Main Program Sweep (Cycle)"
{ S7_Optimized_Access := 'TRUE' }
VERSION : 0.1
   VAR_INPUT
      Initial_Call : Bool;   // Initial call of this OB
      Remanence : Bool;   // =True, if remanent data are available
   END_VAR
BEGIN

REGION Network 1
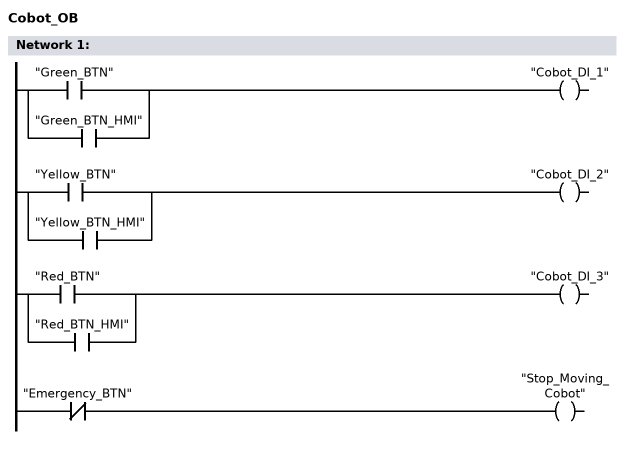
   RUNG wire#powerrail
      Contact( "Green_BTN" )
      wire#w1
      Coil( "Cobot_DI_1" )
   END_RUNG
   RUNG wire#powerrail
      Contact( "Green_BTN_HMI" )
   END_RUNG wire#w1
   RUNG wire#powerrail
      Contact( "Yellow_BTN" )
      wire#w2
      Coil( "Cobot_DI_2" )
   END_RUNG
   RUNG wire#powerrail
      Contact( "Yellow_BTN_HMI" )
   END_RUNG wire#w2
   RUNG wire#powerrail
      Contact( "Red_BTN" )
      wire#w3
      Coil( "Cobot_DI_3" )
   END_RUNG
   RUNG wire#powerrail
      Contact( "Red_BTN_HMI" )
   END_RUNG wire#w3
   RUNG wire#powerrail
      I_Contact( "Emergency_BTN" )
      Coil( "Stop_Moving_Cobot" )
   END_RUNG
   // the same network as SCL:
   "Cobot_DI_1" := "Green_BTN" OR "Green_BTN_HMI";
   "Cobot_DI_2" := "Yellow_BTN" OR "Yellow_BTN_HMI";
   "Cobot_DI_3" := "Red_BTN" OR "Red_BTN_HMI";
   "Stop_Moving_Cobot" := NOT "Emergency_BTN";
END_REGION
END_ORGANIZATION_BLOCK

(* ===== HMI "HMI_RT_1" =====
system functions are stored by id; their names below are inferred from use
connection "HMI_Connection_1": ETHERNET, SMART_S7_1200_OMS

HMI tags "Default tag table"
   "Tag_ScreenNumber" : UInt, internal
   "HMI_BTN1" : Bool = PLC HMI_BTN1 AT %M50.0, 100 ms
   "Conveyor2" : Bool = PLC Conveyor2 AT %Q0.0, 100 ms
   "Pusher1" : Bool = PLC Pusher1 AT %Q0.1, 100 ms
   "Drill" : Bool = PLC Drill AT %Q0.3, 100 ms
   "Mix" : Bool = PLC Mix AT %Q0.5, 100 ms
   "Pusher2" : Bool = PLC Pusher2 AT %Q0.6, 100 ms
   "Conveyor5" : Bool = PLC Conveyor5 AT %Q0.7, 100 ms
   "Conveyor6_OUT" : Bool = PLC Conveyor6_OUT AT %Q8.3, 100 ms
   "Conveyor6_IN" : Bool = PLC Conveyor6_IN AT %Q8.2, 100 ms
   "Red_Tower" : Bool = PLC Red_Tower AT %Q1.1, 100 ms
   "Green_Tower" : Bool = PLC Green_Tower AT %Q1.0, 100 ms
   "cakeFlavor" : UInt = PLC cakeFlavor AT %MW12, 1 s
   "Conveyor3" : Bool = PLC Conveyor3 AT %Q0.2, 100 ms
   "Conveyor4" : Bool = PLC Conveyor4 AT %Q0.4, 100 ms
   "Press_UP" : Bool = PLC Press_UP AT %Q8.4, 100 ms
   "Press_DOWN" : Bool = PLC Press_DOWN AT %Q8.5, 100 ms
   "drillingTime" : Time = PLC drillingTime AT %MD14, 1 s
   "processTimes_DB_chocolateDrillingInput" : UInt = PLC processTimes_DB.chocolateDrillingInput_ms, 1 s
   "processTimes_DB_chocolateMixingInput" : UInt = PLC processTimes_DB.chocolateMixingInput_ms, 1 s
   "processTimes_DB_vanillaDrillingInput_ms" : UInt = PLC processTimes_DB.vanillaDrillingInput_ms, 1 s
   "processTimes_DB_vamillaMixingInput_ms" : UInt = PLC processTimes_DB.vanillaMixingInput_ms, 1 s
   "processTimes_DB_strawberryDrillingInput_ms" : UInt = PLC processTimes_DB.strawberryDrillingInput_ms, 1 s
   "processTimes_DB_strawberryMixingInput_ms" : UInt = PLC processTimes_DB.strawberryMixingInput_ms, 1 s
   "ManualMode_SW" : Bool = PLC ManualMode_SW AT %M53.0, 1 s
   "HMI_BTN_Conveyor2" : Bool = PLC HMI_BTN_Conveyor2 AT %M50.1, 1 s
   "HMI_BTN_Pusher1" : Bool = PLC HMI_BTN_Pusher1 AT %M50.2, 1 s
   "HMI_BTN_Conveyor3" : Bool = PLC HMI_BTN_Conveyor3 AT %M50.3, 1 s
   "HMI_BTN_Conveyor4" : Bool = PLC HMI_BTN_Conveyor4 AT %M50.4, 1 s
   "HMI_BTN_Drill" : Bool = PLC HMI_BTN_Drill AT %M50.6, 1 s
   "HMI_BTN_Mix" : Bool = PLC HMI_BTN_Mix AT %M50.7, 1 s
   "HMI_BTN_Conveyor5" : Bool = PLC HMI_BTN_Conveyor5 AT %M50.5, 1 s
   "HMI_BTN_Pusher2" : Bool = PLC HMI_BTN_Pusher2 AT %M51.0, 1 s

text list "Flavors": 0 'Chocolate'; 1 'Vanilla'; 2 'Strawberry'; 4 'Flavor'

Template "Template_1" 800x480
   Button "Template_Button" at 714,429 size 71x50; TextOff 'Text'
   Button "Template_Button_1" at 614,429 size 71x50; TextOff 'Text'
   Button "Template_Button_2" at 514,429 size 71x50; TextOff 'Text'
   Button "Start screen" at 414,429 size 71x50; TextOff 'Start screen'; PictureOff "NavigateHome_KTP700_Basic_PN_TR"; PictureOn "NavigateHome_KTP700_Basic_PN_TR"
      on Release: ActivateScreen("Root screen", 0)
   Button "Exit" at 314,429 size 71x50; TextOff 'Exit'; PictureOff "ExitRuntime_KTP700_Basic_PN_TR"; PictureOn "ExitRuntime_KTP700_Basic_PN_TR"
      on Release: StopRuntime(0)
   Button "Language" at 214,429 size 71x50; TextOff 'Language'; PictureOff "ToggleLanguage_KTP700_Basic_PN_TR"; PictureOn "ToggleLanguage_KTP700_Basic_PN_TR"
      on Release: function_fb9197e8(-1)
   Button "Log on" at 114,429 size 71x50; TextOff 'Log on'; PictureOff "Login_KTP700_Basic_PN_TR"; PictureOn "Login_KTP700_Basic_PN_TR"
      on Release: function_a2a04561()
   Button "Alarms" at 14,429 size 71x50; TextOff 'Alarms'; PictureOff "AlarmDisplay_KTP700_Basic_PN_TR"; PictureOn "AlarmDisplay_KTP700_Basic_PN_TR"
      on Release: function_ef3f5d25("Alarm window_Unacknowledged", -1)
   SymbolicIOField "Symbolic_IO_Field_Screen" at 53,9 size 640x33; TextOff '0'; TextOn '1'; TextList "TextList_ScreenNames"
      ProcessValue <- "Tag_ScreenNumber"
      on Change: ActivateScreenByNumber("Tag_ScreenNumber", 0)
   DateTimeField "HmiScreenItemData" at 695,25 size 105x25
   DateTimeField "HmiScreenItemData_1" at 695,0 size 105x25
   GraphicView "Logo" at 0,0 size 51x51; Picture "atoleLogo"

screen "Root screen" 800x480, template "Template_1"
   on GenerateScreen: SetTag("Tag_ScreenNumber", 1)
   TextField "HmiScreenItemData" at 40,48 size 720x57; Text 'Welcome to ATOLE S.A. de C.V.'
   Button "Button_1" at 312,336 size 80x40; TextOff 'BTN_1'
      on Press: SetBit("HMI_BTN1")
      on Release: ResetBit("HMI_BTN1")
   Button "Button_2" at 88,224 size 200x40; TextOff 'Plant View'
      on Press: ActivateScreen("PlantView", 0)
   SymbolicIOField "Symbolic I/O field_1" at 88,160 size 200x40; TextOff '0'; TextOn '1'; TextList "Flavors"
      ProcessValue <- "cakeFlavor"
   GraphicView "Graphic view_1" at 464,112 size 294x294; Picture "cake"
   Button "Button_3" at 88,280 size 200x40; TextOff 'Set Process Times'
      on Press: ActivateScreen("ProcessTimes", 0)
   Button "Button_4" at 88,336 size 200x40; TextOff 'Manual Control'
      on Press: ActivateScreen("ManualControl", 0)

screen "PlantView" 800x480
   GraphicView "Graphic view_1" at 14,67 size 773x401; Picture "machiningCellDiagram_2"
   Button "Button_1" at 16,432 size 96x32; TextOff 'Home'
      on Press: ActivateScreen("Root screen", 0)
   Circle "Circle_1" at 684,79 size 11x11
      Visibility <- "Conveyor2"
   Circle "Circle_2" at 747,245 size 11x11
      Visibility <- "Pusher1"
   Circle "Circle_3" at 546,379 size 11x11
      Visibility <- "Drill"
   Circle "Circle_4" at 323,428 size 11x11
      Visibility <- "Pusher2"
   Circle "Circle_5" at 342,137 size 11x11
      Visibility <- "Conveyor5"
   Circle "Circle_6" at 400,379 size 11x11
      Visibility <- "Mix"
   GraphicView "Graphic view_2" at 33,105 size 21x24; Picture "arrow"
      Visibility <- "Conveyor6_OUT"
   GraphicView "Graphic view_3" at 33,179 size 21x24; Picture "arrowDown"
      Visibility <- "Conveyor6_IN"
   Rectangle "Rectangle_1" at 670,353 size 20x20
      Visibility <- "Red_Tower"
   Rectangle "Rectangle_2" at 699,353 size 20x20
      Visibility <- "Green_Tower"
   TextField "Text field_1" at 320,16 size 162x39; Text 'Plant View'
   Circle "Circle_7" at 556,187 size 11x11
      Visibility <- "Conveyor3"
   Circle "Circle_8" at 417,187 size 11x11
      Visibility <- "Conveyor4"
   GraphicView "Graphic view_4" at 33,354 size 21x24; Picture "arrowDown"
      Visibility <- "Press_DOWN"
   GraphicView "Graphic view_5" at 33,279 size 21x24; Picture "arrow"
      Visibility <- "Press_UP"

screen "ManualControl" 800x480
   Switch "Switch_1" at 16,212 size 120x56; CaptionText 'Switch'; TextOff 'OFF'; TextOn 'ON'
      ProcessValue <- "ManualMode_SW"
   Button "Button_1" at 16,432 size 96x32; TextOff 'Home'
      on Press: ActivateScreen("Root screen", 0)
   TextField "Text field_1" at 286,24 size 229x39; Text 'Manual Control'
   Button "Button_2" at 168,88 size 144x32; TextOff 'Conveyor 2'
      on Press: SetBit("HMI_BTN_Conveyor2")
      on Release: ResetBit("HMI_BTN_Conveyor2")
   Button "Button_3" at 168,136 size 144x32; TextOff 'Pusher 1'
      on Press: SetBit("HMI_BTN_Pusher1")
      on Release: ResetBit("HMI_BTN_Pusher1")
   Button "Button_4" at 168,184 size 144x32; TextOff 'Conveyor 3'
      on Release: ResetBit("HMI_BTN_Conveyor3")
      on Press: SetBit("HMI_BTN_Conveyor3")
   Button "Button_5" at 168,232 size 144x32; TextOff 'Conveyor 4'
      on Press: SetBit("HMI_BTN_Conveyor4")
      on Release: ResetBit("HMI_BTN_Conveyor4")
   Button "Button_6" at 168,280 size 144x32; TextOff 'Drill'
      on Press: SetBit("HMI_BTN_Drill")
      on Release: ResetBit("HMI_BTN_Drill")
   Button "Button_7" at 168,328 size 144x32; TextOff 'Mix'
      on Press: SetBit("HMI_BTN_Mix")
      on Release: ResetBit("HMI_BTN_Mix")
   Button "Button_8" at 168,376 size 144x32; TextOff 'Pusher 2'
      on Press: SetBit("HMI_BTN_Pusher2")
      on Release: ResetBit("HMI_BTN_Pusher2")
   Button "Button_9" at 168,424 size 144x32; TextOff 'Conveyor 5'
      on Press: SetBit("HMI_BTN_Conveyor5")
      on Release: ResetBit("HMI_BTN_Conveyor5")

screen "ProcessTimes" 800x480
   TextField "Text field_1" at 294,16 size 213x39; Text 'Process Times'
   IOField "I/O field_1" at 120,192 size 152x48; FormatPattern 9999999; Unit  s
      ProcessValue <- "processTimes_DB_chocolateDrillingInput"
   IOField "I/O field_2" at 120,264 size 152x48; FormatPattern 9999999; Unit  s
      ProcessValue <- "processTimes_DB_chocolateMixingInput"
   TextField "Text field_2" at 152,168 size 86x23; Text 'Chocolate'
   TextField "Text field_3" at 408,168 size 61x23; Text 'Vanilla'
   TextField "Text field_4" at 624,168 size 96x23; Text 'Strawberry'
   IOField "I/O field_3" at 360,264 size 152x48; FormatPattern 9999999; Unit  s
      ProcessValue <- "processTimes_DB_vamillaMixingInput_ms"
   IOField "I/O field_4" at 360,192 size 152x48; FormatPattern 9999999; Unit  s
      ProcessValue <- "processTimes_DB_vanillaDrillingInput_ms"
   IOField "I/O field_5" at 600,192 size 152x48; FormatPattern 9999999; Unit  s
      ProcessValue <- "processTimes_DB_strawberryDrillingInput_ms"
   IOField "I/O field_6" at 600,264 size 152x48; FormatPattern 9999999; Unit  s
      ProcessValue <- "processTimes_DB_strawberryMixingInput_ms"
   TextField "Text field_5" at 24,200 size 64x23; Text 'Drilling'
   TextField "Text field_6" at 24,272 size 59x23; Text 'Mixing'
   Button "Button_1" at 16,432 size 96x32; TextOff 'Home'
      on Press: ActivateScreen("Root screen", 0)
*)

(* ===== HMI "HMI_RT_2" =====
system functions are stored by id; their names below are inferred from use
connection "HMI_Connection_2": ETHERNET, SMART_S7_1200_OMS

HMI tags "Default tag table"
   "Tag_ScreenNumber" : UInt, internal
   "Vertical_Piston" : Bool = PLC Vertical_Piston AT %Q8.5, 1 s

Template "Template_1" 800x480
   Button "Template_Button" at 714,429 size 71x50; TextOff 'Text'
   Button "Template_Button_1" at 614,429 size 71x50; TextOff 'Text'
   Button "Template_Button_2" at 514,429 size 71x50; TextOff 'Text'
   Button "Start screen" at 414,429 size 71x50; TextOff 'Start screen'; PictureOff "NavigateHome_KTP700_Basic_PN_TR"; PictureOn "NavigateHome_KTP700_Basic_PN_TR"
      on Release: ActivateScreen("Root screen", 0)
   Button "Exit" at 314,429 size 71x50; TextOff 'Exit'; PictureOff "ExitRuntime_KTP700_Basic_PN_TR"; PictureOn "ExitRuntime_KTP700_Basic_PN_TR"
      on Release: StopRuntime(0)
   Button "Language" at 214,429 size 71x50; TextOff 'Language'; PictureOff "ToggleLanguage_KTP700_Basic_PN_TR"; PictureOn "ToggleLanguage_KTP700_Basic_PN_TR"
      on Release: function_fb9197e8(-1)
   Button "Log on" at 114,429 size 71x50; TextOff 'Log on'; PictureOff "Login_KTP700_Basic_PN_TR"; PictureOn "Login_KTP700_Basic_PN_TR"
      on Release: function_a2a04561()
   Button "Alarms" at 14,429 size 71x50; TextOff 'Alarms'; PictureOff "AlarmDisplay_KTP700_Basic_PN_TR"; PictureOn "AlarmDisplay_KTP700_Basic_PN_TR"
      on Release: function_ef3f5d25("Alarm window_Unacknowledged", -1)
   SymbolicIOField "Symbolic_IO_Field_Screen" at 53,9 size 640x33; TextOff '0'; TextOn '1'; TextList "TextList_ScreenNames"
      ProcessValue <- "Tag_ScreenNumber"
      on Change: ActivateScreenByNumber("Tag_ScreenNumber", 0)
   DateTimeField "HmiScreenItemData" at 695,25 size 105x25
   DateTimeField "HmiScreenItemData_1" at 695,0 size 105x25
   GraphicView "Logo" at 0,0 size 51x51; Picture "Logo of HMI_2"

screen "Root screen" 800x480, template "Template_1"
   on GenerateScreen: SetTag("Tag_ScreenNumber", 1)
   TextField "HmiScreenItemData" at 40,48 size 720x57; Text 'Welcome to ATOLE S.A. de C.V.'
   GraphicView "Graphic view_1" at 464,112 size 294x294; Picture "strawberryCake"
   Button "Button_2" at 159,191 size 200x40; TextOff 'Plant View'
      on Press: ActivateScreen("Pneumatic_Monitoring", 0)
   Button "Button_3" at 159,247 size 200x40; TextOff 'Set Process Times'
      on Press: ActivateScreen("ProcessTimes", 0)
   Button "Button_4" at 159,303 size 200x40; TextOff 'Manual Control'
      on Press: ActivateScreen("ManualControl", 0)

screen "Pneumatic_Monitoring" 800x480
   TextField "Text field_1" at 320,16 size 162x39; Text 'Plant View'
   Button "Button_1" at 16,432 size 96x32; TextOff 'Home'
      on Press: ActivateScreen("Root screen", 0)
   GraphicView "Graphic view_1" at 111,77 size 593x386; Picture "pneumaticCellDiagram"
*)